Staubli VAL3: simpleCommTest.pjx

--- simpleCommTest.pjx ---
Parameters version=s7.7.2 stackSize=5000 millimeterUnit=true
Program file=recvData.pgx
Program file=sendData.pgx
Program file=start.pgx
Program file=stop.pgx
Data file=simpleCommTest.dtx

--- simpleCommTest.dtx ---
public bool bReceiver
public bool bSender
mdesc mNomSpeed
public num n
public num nB = -1
public num nByteIn[24]
public num nByteOut[24]
public num nTrsfIn[6]
public num nTrsfOut[6]
public sio siTcpReceiver = {link=Socket\Feedback}
public sio siTcpSender = {link=Socket\Motion}
public trsf trShiftIn
public trsf trShiftOut

--- start.pgx ---
program start()
begin
  taskCreateSync "sender",0.5,bSender,sendData()
  taskCreateSync "receiver",0.5,bReceiver,recvData()
end

--- recvData.pgx ---
public program recvData()
begin
  while (true)
    nB=0
    n=0
    while (nB<24)
      nB=sioGet(siTcpReceiver,nByteIn[n])
      if (nB>0)
        n=n+nB
      else
        // communication error
        popUpMsg("Comm error")
        return
      endIf
    endWhile
    if (fromBinary(nByteIn,24,"-4l",nTrsfIn)!=6)
      // corrupted data
      popUpMsg("Data corrupted")
      return
    else
      trShiftIn.x=nTrsfIn[0]
      trShiftIn.y=nTrsfIn[1]
      trShiftIn.z=nTrsfIn[2]
      trShiftIn.rx=nTrsfIn[3]
      trShiftIn.ry=nTrsfIn[4]
      trShiftIn.rz=nTrsfIn[5]
    endIf
  endWhile
end

--- sendData.pgx ---
public program sendData()
  local num l_nRetVal
begin
  userPage()
  while (true)
    nTrsfOut[0]=trShiftOut.x
    nTrsfOut[1]=trShiftOut.y
    nTrsfOut[2]=trShiftOut.z
    nTrsfOut[3]=trShiftOut.rx
    nTrsfOut[4]=trShiftOut.ry
    nTrsfOut[5]=trShiftOut.rz

    toBinary(nTrsfOut,6,"-4l",nByteOut)
    l_nRetVal = sioSet(siTcpSender,nByteOut)
    if (l_nRetVal == -1)
      putln("Not connected")
    endIf
  endWhile
end

--- stop.pgx ---
program stop()
begin
end
